% RSLogix 500 project BASI INPUT OUTPUT.RSS, saved by version 8.30.00.16 %
PROJECT ""    % processor: Bul.1763 MicroLogix 1100 Series B %

PROGRAM FILES
  LAD 2 "AIN"  4 rungs
  LAD 3 "ALAR"  1 rungs
  LAD 4 "DIGITAL IO"  3 rungs  % INPUTS OUTPUTS %
  LAD 5 "ANALOG IO"  2 rungs

DATA FILES
  O0 OUTPUT  7 elements
  I1 INPUT  13 elements
  S2 STATUS  66 elements
  B3 BINARY  10 elements
  T4 TIMER  1 elements
  C5 COUNTER  1 elements
  R6 CONTROL  1 elements
  N7 INTEGER  1 elements
  F8 FLOAT  1 elements

LADDER 2 "AIN"
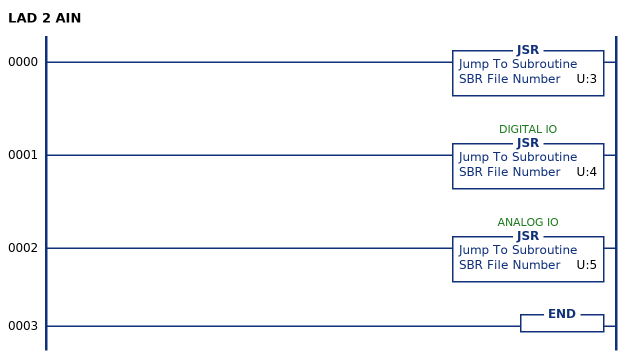
% Rung: 0 %
SOR JSR U:3 EOR
% Rung: 1 %
SOR JSR U:4 EOR
%   U:4  "DIGITAL IO" %
% Rung: 2 %
SOR JSR U:5 EOR
%   U:5  "ANALOG IO" %
% Rung: 3 %
SOR END EOR

LADDER 4 "DIGITAL IO"    % INPUTS OUTPUTS %
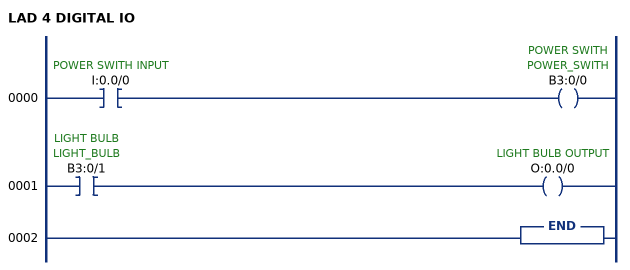
% Rung: 0 %
SOR XIC I:0.0/0 OTE B3:0/0 EOR
%   I:0.0/0  "POWER SWITH INPUT" %
%   B3:0/0  POWER_SWITH  "POWER SWITH" %
% Rung: 1 %
SOR XIC B3:0/1 OTE O:0.0/0 EOR
%   B3:0/1  LIGHT_BULB  "LIGHT BULB" %
%   O:0.0/0  "LIGHT BULB OUTPUT" %
% Rung: 2 %
SOR END EOR

LADDER 5 "ANALOG IO"
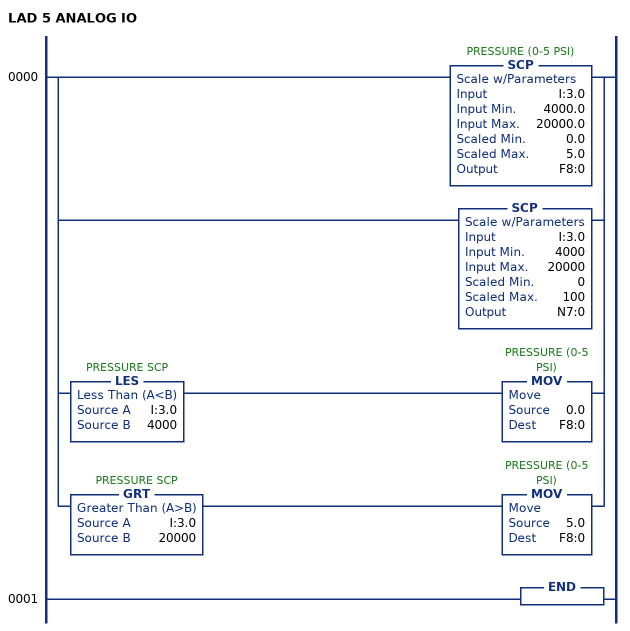
% Rung: 0 %
SOR BST SCP I:3.0 4000.0 20000.0 0.0 5.0 F8:0 NXB SCP I:3.0 4000 20000 0 100 N7:0 NXB LES I:3.0 4000 MOV 0.0 F8:0 NXB GRT I:3.0 20000 MOV 5.0 F8:0 BND EOR
%   I:3.0  SCP  "PRESSURE" %
%   F8:0  "PRESSURE (0-5 PSI)" %
% Rung: 1 %
SOR END EOR

OTHER DOCUMENTED ADDRESSES
  O:0.0/5  MOVE_EDGE_RIGHT
  O:0.0/6  MOVE_EDGE_LEFT
  PFILE:3  "Emergency and enable push buttons"

DATA TABLE (non-zero values as saved)
DATA B3
% B3:0 % 0X0001 0X0000 0X0000 0X0000 0X0000 0X0000 0X0000 0X0000 0X0000 0X0000
